% RSLogix 500 project I2P JOB 13 A - SOLUTION.RSS, saved by version 10.00.00.00 %
PROJECT "ML01A"    % processor: Bul.1763 MicroLogix 1100 Series B %

PROGRAM FILES
  LAD 2   9 rungs

DATA FILES
  O0 OUTPUT  4 elements
  I1 INPUT  6 elements
  S2 STATUS  66 elements
  B3 BINARY  1 elements
  T4 TIMER  1 elements
  C5 COUNTER  1 elements
  R6 CONTROL  1 elements
  N7 INTEGER  1 elements
  F8 FLOAT  1 elements

LADDER 2
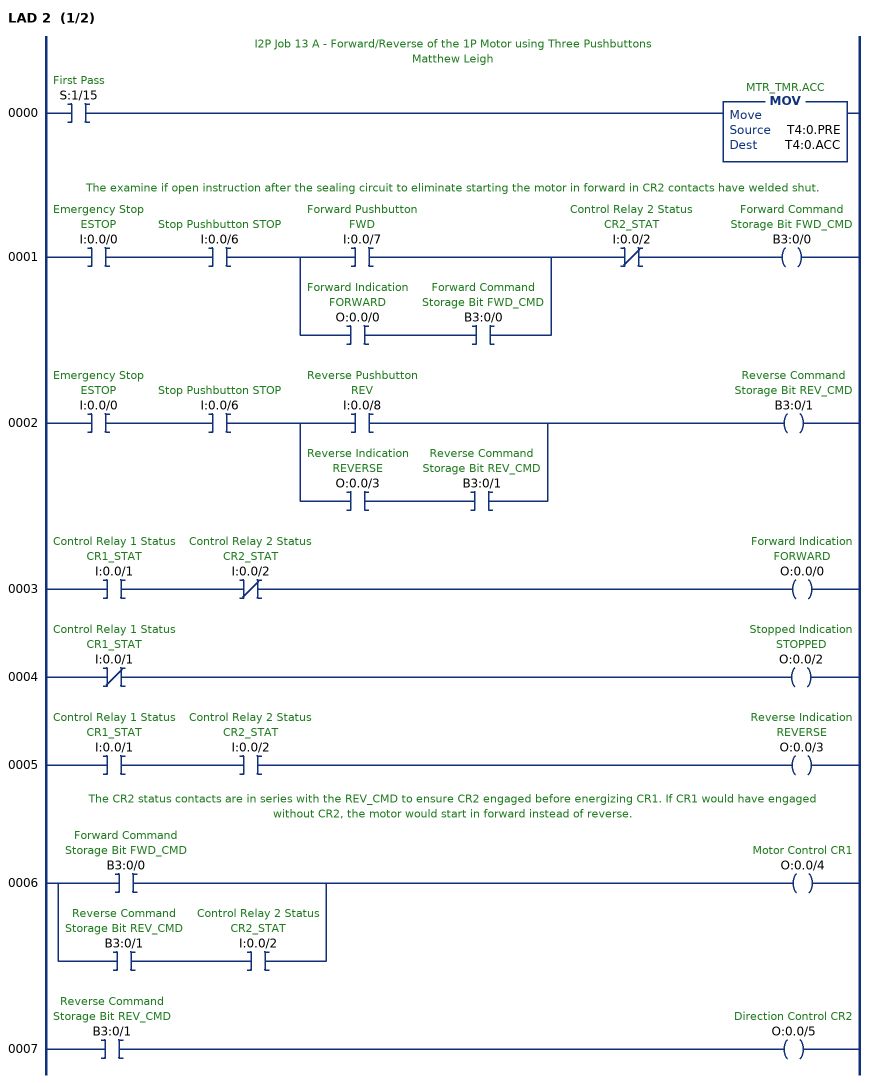
% Rung: 0 %
% I2P Job 13 A - Forward/Reverse of the 1P Motor using Three Pushbuttons
% Matthew Leigh %
SOR XIC S:1/15 MOV T4:0.PRE T4:0.ACC EOR
%   S:1/15  "First Pass" %
%   T4:0  MTR_TMR %
% Rung: 1 %
% The examine if open instruction after the sealing circuit to eliminate starting the motor in forward in CR2 contacts have welded shut. %
SOR XIC I:0.0/0 XIC I:0.0/6 BST XIC I:0.0/7 NXB XIC O:0.0/0 XIC B3:0/0 BND XIO I:0.0/2 OTE B3:0/0 EOR
%   I:0.0/0  ESTOP  "Emergency Stop" %
%   I:0.0/6  STOP  "Stop Pushbutton" %
%   I:0.0/7  FWD  "Forward Pushbutton" %
%   O:0.0/0  FORWARD  "Forward Indication" %
%   B3:0/0  FWD_CMD  "Forward Command Storage Bit" %
%   I:0.0/2  CR2_STAT  "Control Relay 2 Status" %
% Rung: 2 %
SOR XIC I:0.0/0 XIC I:0.0/6 BST XIC I:0.0/8 NXB XIC O:0.0/3 XIC B3:0/1 BND OTE B3:0/1 EOR
%   I:0.0/0  ESTOP  "Emergency Stop" %
%   I:0.0/6  STOP  "Stop Pushbutton" %
%   I:0.0/8  REV  "Reverse Pushbutton" %
%   O:0.0/3  REVERSE  "Reverse Indication" %
%   B3:0/1  REV_CMD  "Reverse Command Storage Bit" %
% Rung: 3 %
SOR XIC I:0.0/1 XIO I:0.0/2 OTE O:0.0/0 EOR
%   I:0.0/1  CR1_STAT  "Control Relay 1 Status" %
%   I:0.0/2  CR2_STAT  "Control Relay 2 Status" %
%   O:0.0/0  FORWARD  "Forward Indication" %
% Rung: 4 %
SOR XIO I:0.0/1 OTE O:0.0/2 EOR
%   I:0.0/1  CR1_STAT  "Control Relay 1 Status" %
%   O:0.0/2  STOPPED  "Stopped Indication" %
% Rung: 5 %
SOR XIC I:0.0/1 XIC I:0.0/2 OTE O:0.0/3 EOR
%   I:0.0/1  CR1_STAT  "Control Relay 1 Status" %
%   I:0.0/2  CR2_STAT  "Control Relay 2 Status" %
%   O:0.0/3  REVERSE  "Reverse Indication" %
% Rung: 6 %
% The CR2 status contacts are in series with the REV_CMD to ensure CR2 engaged before energizing CR1. If CR1 would have engaged without CR2, the motor would start in forward instead of reverse. %
SOR BST XIC B3:0/0 NXB XIC B3:0/1 XIC I:0.0/2 BND OTE O:0.0/4 EOR
%   B3:0/0  FWD_CMD  "Forward Command Storage Bit" %
%   B3:0/1  REV_CMD  "Reverse Command Storage Bit" %
%   I:0.0/2  CR2_STAT  "Control Relay 2 Status" %
%   O:0.0/4  CR1  "Motor Control" %
% Rung: 7 %
SOR XIC B3:0/1 OTE O:0.0/5 EOR
%   B3:0/1  REV_CMD  "Reverse Command Storage Bit" %
%   O:0.0/5  CR2  "Direction Control" %

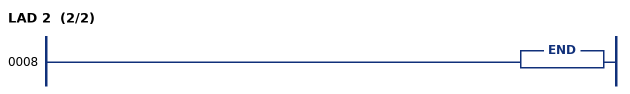
% Rung: 8 %
SOR END EOR

OTHER DOCUMENTED ADDRESSES
  B3:0/2  LAST_FWD  "Last Direction was Forward"
  B3:0/3  LAST_REV  "Last Direction was Reverse"
  B3:0/4  DIR_CHNG  "Direction Change Indication"
  O:0.0/1  WAIT  "Wait for Start Switch"

DATA TABLE (non-zero values as saved)
DATA T4
% .PRE .ACC %
% T4:0 % 8 0
